ABB RobotStudio station: Project1.rsstnx

Station Project1 (saved by RobotStudio 22.3.10141.1)
Controller Controlador1, task T_ROB1: task frame (RAPID world) sits at (500, 500, 0) mm, rotated rx 0 ry 0 rz 180 deg in the station
Controller Controlador1
  mechanical unit ROB_1: IRB120_3_58__01, 6 joints, base frame (0, 0, 0) mm
Layout (positions relative to the parent item):
  - IRB120_3_58__01 [mechanism, from Robots\IRB120_3_58_G_01.rslib] at (500, 500, 0) mm, rotated rx 0 ry 0 rz 180 deg; joint values [1.7542, 0.156, -0.3304, 0.2848, 1.629, 0] (rad or m)
  - table_and_fixture_140 [part, from Training Objects\propeller_table.rslib]
